// TIA Portal V17 export
// export: Created 2024-08-09T12:53:15.1931795Z, ExportSetting WithDefaults, DisplayName Totally Integrated Automation Portal, DisplayVersion V17 Update 7, DisplayName TIA Portal Openness, DisplayVersion V17 Update 7, DisplayName TIA Portal Version Control Interface, DisplayVersion V17, DisplayName STEP 7 Professional, DisplayVersion V17 Update 7, DisplayName STEP 7 Safety, DisplayVersion V17 Update 6, DisplayName WinCC Professional, DisplayVersion V17 Update 7
VAR_GLOBAL   // PLC tag table "Dec_Niveaux_Chpont"
END_VAR
VAR_GLOBAL CONSTANT   // user constants
   ChPont_AttDemCir_Niv : USInt := 10;
   ChPont_DemCir_Niv : USInt := 20;
   ChPont_CircuitPret_Niv : USInt := 30;
   ChPont_ChargEc_Niv : USInt := 40;
   ChPont_ConfFinCharg_Niv : USInt := 50;
   ChPont_VidCir_Niv : USInt := 60;
   ChPont_FVidCir_Niv : USInt := 160;
   ChPont_FinLot_Niv : USInt := 255;
END_VAR
